	242: // Adding mover to group
		bWatchDogActive := TRUE;
		THIS^.fbMoversPresent.ResetIterator();
		WHILE THIS^.fbMoversPresent.HasNextObject() DO
			IF ToXpMover(THIS^.fbMoversPresent.GetNextObject(),ipTempMover) THEN
				hr := GetMostSignificant(hr, ipTempMover.Feedback.HR);
			END_IF
		END_WHILE
		
		IF CheckOk(hr) THEN 
			nSeqEnabling := 300;
		ELSIF FAILED(hr) THEN
			nSeqEnabling := 1000 + nSeqEnabling;
		END_IF		
	
		
		
	300: // Enable group
		bWatchDogActive := TRUE;
		hr := ipGroup.Enable();
		
		IF CheckOk(hr) THEN 
			nSeqEnabling := 310;
		ELSE
			nSeqEnabling := 1000 + nSeqEnabling;
		END_IF	
		
	310: // Enabling group
		bWatchDogActive := TRUE;
		hr := ipGroup.Feedback.HR;
		
		IF CheckOk(hr) THEN 
			//nSeqEnabling := 350;
			nSeqEnabling := 400;
		ELSIF FAILED(hr) THEN
			nSeqEnabling := 1000 + nSeqEnabling;
		END_IF	
		
		
//	340: // Check dist last known position to current pos
//		bWatchDogActive := TRUE;
//		THIS^.fbMovers.ResetIterator();
//		WHILE THIS^.fbMovers.HasNextObject() DO
//			IF ToXpMover(THIS^.fbMovers.GetNextObject(),ipTempMover) THEN
//				IF ipTempMover.PositionAtDisable.x <> 0 AND ipTempMover.PositionAtDisable.y <> 0 THEN
//					fDistLastToSet := F_DistXYVectors(ipTempMover.PositionAtDisable, ipTempMover.PositionSet);
//					fMaxError := MAX(fMaxError, fDistLastToSet);
//				END_IF
//			END_IF
//		END_WHILE
//		IF fMaxError < 50 THEN
//			nSeqEnabling := 350;
//		ELSE
//			nSeqEnabling := 400;			
//		END_IF
//
//		
//	350: // Move to last valide known position
//		bWatchDogActive := TRUE;
//		THIS^.fbMovers.ResetIterator();
//		WHILE THIS^.fbMovers.HasNextObject() DO
//			IF ToXpMover(THIS^.fbMovers.GetNextObject(),ipTempMover) THEN
//				IF ipTempMover.PositionAtDisable.x <> 0 AND ipTempMover.PositionAtDisable.y <> 0 THEN
//					hr := GetMostSignificant(hr, ipTempMover.MoveXY(fPosition_X := ipTempMover.PositionAtDisable.x, 
//																	fPosition_Y := ipTempMover.PositionAtDisable.y));
//				END_IF
//			END_IF
//		END_WHILE
//		//Its posible that the command failed. Do not exit SEQ
//		nSeqEnabling := 351;
//
//
//		
//	351: // Wait for standstill
//		bWatchDogActive := TRUE;
//		
//		bOk := TRUE;
//		THIS^.fbMovers.ResetIterator();
//		WHILE THIS^.fbMovers.HasNextObject() DO
//			IF ToXpMover(THIS^.fbMovers.GetNextObject(),ipTempMover) THEN
//				bOk := bOk AND ipTempMover.Standstill;
//			END_IF
//		END_WHILE
//		THIS^.fbMovers.RestoreIterator();
//		
//		IF bOk THEN 
//			nSeqEnabling := 400;
//		END_IF	

		
	400: (*	Restart of the sequenze "JoiningTrack". Default strategy is that each mover joins the closest track
			Outsourced to a method for easier overwriting *)
		THIS^.nSeqJoiningTrack := 0;	
		nSeqEnabling := 401;
	

	401: (*	Default strategy is that each mover joins the closest track
			Outsourced to a method for easier overwriting *)
		hr := THIS^.JoiningTrack();

		IF CheckOk(hr) THEN 
			nSeqEnabling := 500;
		ELSIF FAILED(hr) THEN
			nSeqEnabling := 1000 + nSeqEnabling;
		END_IF	
		
	

	
	500: (*	Restart of the sequenze "JoiningStation" to distribute the movers to the available stations.
			Outsourced to a method for easier overwriting *)
		THIS^.nSeqJoiningStation := 0;	
		nSeqEnabling := 501;	
	
	501: (*	Distribute the movers to the available stations.
		 	Outsourced to a method for easier overwriting *)
		hr := THIS^.JoiningStation();

		IF CheckOk(hr) THEN 
			nSeqEnabling := SEQ_DONE;
		ELSIF FAILED(hr) THEN
			nSeqEnabling := 1000 + nSeqEnabling;
		END_IF	

		
	SEQ_DONE: // Done
		Enabling := S_OK;

		
	1000..1999://Error
		hr := GetMostSignificant(hrLastCycle, E_FAIL);
		//Only rais if timeout is not active
		IF NOT fbErrorEnabling.bRaised AND NOT fbTimeOutEnabling.bRaised THEN 
			fbErrorEnabling.CreateEx(stEventEntry:=TC_EVENTS.CHALET_Base_Events.ErrorEnabling, ipSourceInfo := THIS^.fbSourceInfo, bWithConfirmation := FALSE);
			fbErrorEnabling.ipArguments.AddUInt(nSeqEnabling-1000);
			fbErrorEnabling.Raise(0);
		END_IF
	
	ELSE
		//Timeout unknown state
		bWatchDogActive := TRUE;
END_CASE


//Timeout after to long stay in one of the following seq.
fbTimeOutSeq.IN := (nlastState = nSeqEnabling) AND bWatchDogActive;
fbTimeOutSeq.PT := TO_TIME(XPlanarParameterlist.F_TIMEOUT_ERROR_ENABLING*1000.0);
fbTimeOutSeq();
nlastState := nSeqEnabling;

IF fbTimeOutSeq.Q THEN
	IF NOT fbTimeOutEnabling.bRaised THEN 
		fbTimeOutEnabling.CreateEx(stEventEntry:=TC_EVENTS.CHALET_Base_Events.TimeOutEnabling, ipSourceInfo := THIS^.fbSourceInfo, bWithConfirmation := FALSE);
		fbTimeOutEnabling.ipArguments.AddUInt(nSeqEnabling);
		fbTimeOutEnabling.Raise(0);
	END_IF
	//next seq is error
	nSeqEnabling := 1000 + nSeqEnabling;
END_IF

//Clear Tc3-Eventlogger alarm 
IF nSeqEnabling <= SEQ_DONE THEN
	fbTimeOutEnabling.Clear(0,0);
	fbErrorEnabling.Clear(0,0);
	fbErrorMoverDetection.Clear(0,0);
END_IF


//store last information
hrLastCycle := hr;

// Propagate error
IF FAILED(hr) THEN
	Enabling := hr;
END_IF
END_METHOD

{attribute 'monitoring':='call'}
PROPERTY Enviroment : I_XP_Environment
GET
Enviroment := THIS^.ipEnvironment;
END_GET
END_PROPERTY

METHOD FastStop : I_CH_Feedback
VAR
	ipMoverPlc : I_XP_Mover_PLC;
END_VAR
THIS^.MoversPresent.ResetIterator();
WHILE THIS^.MoversPresent.HasNextObject() DO
	IF __QUERYINTERFACE(THIS^.MoversPresent.GetNextObject(),ipMoverPlc) THEN
		//Change deceleration to MC_MAXIMUM for each mover
		ipMoverPlc.SetDynConstraint_Path(V:= MC_DEFAULT, A:= MC_DEFAULT, D:= MC_MAXIMUM, J:= MC_MAXIMUM);
	END_IF
END_WHILE
THIS^.MoversPresent.RestoreIterator();


FastStop := THIS^.Disable();
THIS^.Disabling();
END_METHOD

METHOD FB_init : BOOL
VAR_INPUT
	bInitRetains : BOOL; // if TRUE, the retain variables are initialized (warm start / cold start)
	bInCopyCode : BOOL;  // if TRUE, the instance afterwards gets moved into the copy code (online change)
	
END_VAR
VAR
	fbGetCurTaskIdx  : GETCURTASKINDEX;
END_VAR
THIS^.fbFeedback.ActiveCommand 		:= TO_STRING(THIS^.eActiveCommand);
END_METHOD

{attribute 'monitoring':='call'}
PROPERTY Feedback : CHALET_BaseComponents.I_CH_Feedback
GET
Feedback := THIS^.fbFeedback;
END_GET
END_PROPERTY

//Returns the station that is closest to the point according to Phytagoras
METHOD GetStationClosestTo : I_XP_Station
VAR_INPUT
	pos : MoverVector;
END_VAR
VAR
	stPositionStation : MoverVector;
	ipEachStation : I_XP_Station;
	fTempDist : LREAL;
	fDistClosestStation: LREAL := CHALET_BaseComponents.GVL_Datatypes.cMaxLreal;
END_VAR
THIS^.fbStationsUsed.ResetIterator();
WHILE THIS^.fbStationsUsed.HasNextObject() DO
	IF __QUERYINTERFACE(THIS^.fbStationsUsed.GetNextObject(),ipEachStation) THEN
		stPositionStation.x := ipEachStation.PositionOnTrackXY.x;
		stPositionStation.y := ipEachStation.PositionOnTrackXY.y;
		
		fTempDist := F_DistXYVectors(pos, stPositionStation);
		
		IF fTempDist <= fDistClosestStation THEN
			fDistClosestStation := fTempDist;
			GetStationClosestTo := ipEachStation;
		END_IF
		
	END_IF
END_WHILE
THIS^.fbStationsUsed.RestoreIterator();
END_METHOD

METHOD Initialize : HRESULT
VAR_INPUT
END_VAR
VAR
	hr 				: HRESULT := S_OK;
	ipEachStation 	: I_XP_Station;
END_VAR
VAR_INST
	//This error cannot be reset. Requires a reset cold
	{attribute 'hide'}	
	fbInitError : FB_TcAlarm;
	{attribute 'hide'}	
	fbMissingInterfaceAlarm : FB_TcAlarm;

END_VAR
//Set to busy on first call
IF THIS^.eActiveCommand <> CHALET_NC.E_NcAxisCommands.Initialize THEN
	THIS^.eActiveCommand 					:= CHALET_NC.E_NcAxisCommands.Initialize;
	THIS^.fbFeedback.ActiveCommand 			:= TO_STRING(THIS^.eActiveCommand);	
	THIS^.fbFeedback.LastCommandAccepted	:= TRUE;		
	THIS^.fbFeedback.Busy 					:= TRUE;
END_IF

//Check Error during FB_Init
IF THIS^.bErrorDuringFbInit THEN
	IF NOT fbInitError.bRaised THEN 
		//This error cannot be reset. Requires a reset cold
		fbInitError.CreateEx(stEventEntry:=TC_EVENTS.CHALET_Base_Events.ErrorFBinit, ipSourceInfo := THIS^.fbSourceInfo, bWithConfirmation := FALSE);
		fbInitError.Raise(0);
	END_IF
	Initialize:= E_FAIL;
	THIS^.fbFeedback.HR := Initialize;
	RETURN;
END_IF	


//Check if Envirement and Group is existing
IF  THIS^.ipGroup = 0 THEN
	IF NOT fbMissingInterfaceAlarm.bRaised THEN 
		//This error cannot be reset. Requires a reset cold
		fbMissingInterfaceAlarm.CreateEx(stEventEntry:=TC_EVENTS.CHALET_XPlanar_Events.MissingGroupe, ipSourceInfo := THIS^.fbSourceInfo, bWithConfirmation := FALSE);
		fbMissingInterfaceAlarm.Raise(0);
	END_IF
	Initialize := E_FAIL;
	THIS^.fbFeedback.HR := Initialize;
	RETURN;
END_IF

//Check if Envirement and Group is existing
IF THIS^.ipEnvironment = 0 THEN
	IF NOT fbMissingInterfaceAlarm.bRaised THEN 
		//This error cannot be reset. Requires a reset cold
		fbMissingInterfaceAlarm.CreateEx(stEventEntry:=TC_EVENTS.CHALET_XPlanar_Events.MissingEnvironment, ipSourceInfo := THIS^.fbSourceInfo, bWithConfirmation := FALSE);
		fbMissingInterfaceAlarm.Raise(0);
	END_IF
	Initialize := E_FAIL;
	THIS^.fbFeedback.HR := Initialize;
	RETURN;
END_IF



//Init envirement first to get access to XPlanar_Utility
IF THIS^.ipEnvironment.Initialize() = S_OK THEN
	hr := GetMostSignificant(hr, THIS^.ipGroup.Initialize());
	hr := GetMostSignificant(hr, THIS^.fbMoversPresent.Initialize());
	hr := GetMostSignificant(hr, THIS^.fbTracks.Initialize());
	hr := GetMostSignificant(hr, THIS^.fbStationsAll.Initialize());
	hr := GetMostSignificant(hr, THIS^.fbTriggers.Initialize());
	hr := GetMostSignificant(hr, THIS^.fbZones.Initialize());
ELSE
	hr := S_PENDING;
END_IF	



THIS^.bInitDone := (hr = S_OK);

Initialize:= hr;

THIS^.fbFeedback.HR := Initialize;
END_METHOD

{attribute 'monitoring':='call'}
PROPERTY Initialized : BOOL
GET
Initialized := bInitDone;
END_GET
END_PROPERTY

METHOD PROTECTED JoiningStation : HRESULT
VAR
	hr : HRESULT;
	ipEachMover : I_XP_Mover;
	ipEachMoverPlc : I_XP_Mover_PLC;
	ipEachMoverInStation : I_XP_Mover;
	ipEachStation : I_XP_Station;
	ipFirstStation : I_XP_Station;
	ipParentStation : I_XP_Station;
	ipTempMoverPlc : I_XP_Mover_PLC;

	//during move on track
	fVelo	: Tc3_Mc3Definitions.MC_LREAL := Tc3_Mc3Definitions.MC_DEFAULT; 
	fAccDec	: Tc3_Mc3Definitions.MC_LREAL := Tc3_Mc3Definitions.MC_DEFAULT;
	bError : BOOL;
	bFound : BOOL;
	bMoverAtCmdPos : BOOL;
	refPosition : REFERENCE TO MoverVector;
	fCalcualtedGapAtMoverPosition : LREAL;

	ipClosestStation : I_XP_Station;
	fDistToStation : LREAL := CHALET_BaseComponents.GVL_Datatypes.cMaxLreal;
END_VAR
VAR_INST
	bResetMovers : BOOL;	

	{attribute 'hide'}	
	fbDelayJoiningStation : TON;
END_VAR
CASE nSeqJoiningStation OF

	0: //Init
		fbDelayJoiningStation.IN := FALSE;
		
		IF fbStationsUsed.IsEmpty THEN
			nSeqJoiningStation := SEQ_DONE;
		ELSE
			nSeqJoiningStation := 10;
		END_IF
	


	
		
	10:	// For each Mover, Clear planed route to target. After enabling the tracks may have change and are not longer existing.
		THIS^.fbMoversPresent.ResetIterator();
		WHILE THIS^.fbMoversPresent.HasNextObject() DO
			IF __QUERYINTERFACE(THIS^.fbMoversPresent.GetNextObject(), ipEachMover) THEN
				//clear route
				ipEachMover.SetRouteToParent(0);
			END_IF
		END_WHILE
		THIS^.fbMoversPresent.RestoreIterator();
		
		//Empty Mover queue in station
		THIS^.fbStationsUsed.ResetIterator();
		WHILE THIS^.fbStationsUsed.HasNextObject() DO
			IF __QUERYINTERFACE(THIS^.fbStationsUsed.GetNextObject(), ipEachStation) THEN
				ipEachStation.DeleteMoversQueue(); // This is also reset the parent of each mover
			END_IF
		END_WHILE
		THIS^.fbStationsUsed.RestoreIterator();
		
		nSeqJoiningStation := 20;
	
	


	
		
	20: (*Check whether the last set station parent (station responsible for continuing to send the mover) is still valid. This is not the case if, for example:
		- Mover was manually moved to a new position
		- Track layout has changed
		- Position of the station has changed - No longer exists	*)
		THIS^.fbMoversPresent.ResetIterator();
		WHILE THIS^.fbMoversPresent.HasNextObject() DO
			IF __QUERYINTERFACE(THIS^.fbMoversPresent.GetNextObject(), ipEachMover) THEN
				//Prio 1: If the station ahead was the parent, kept this as parent. Easily accessible without issues with collision prevention
				ipParentStation := ipEachMover.CurrentTrack.StationAhedPosition(ipEachMover.PositionOnTrack);
				IF ipEachMover.LastValidParentStation = ipParentStation AND ipParentStation <> 0 THEN
					//Set as new parent
					ipParentStation.AddMoverToQueue(ipEachMover);
					CONTINUE; //Check next mover
				END_IF
				
				//Prio 2: If the station closest was the parent, +/- 10mm . Maybe mall issues with collision prevention
				ipParentStation := ipEachMover.CurrentTrack.StationClosestTo(ipEachMover.PositionOnTrack);
				fDistToStation := F_DistXYVectors(ipParentStation.PositionOnTrackXYZABC, ipEachMover.PositionSet);
				IF ipEachMover.LastValidParentStation = ipParentStation AND ipParentStation <> 0 AND fDistToStation < 10.0 THEN
					//Set as new parent
					ipParentStation.AddMoverToQueue(ipEachMover);
					CONTINUE; //Check next mover
				END_IF
				
				//Prio 3: Get any station ahead current position
				ipParentStation := ipEachMover.CurrentTrack.StationAhedPosition(ipEachMover.PositionOnTrack);
				//Set as new parent
				ipParentStation.AddMoverToQueue(ipEachMover);
			END_IF
		END_WHILE
		THIS^.fbMoversPresent.RestoreIterator();	
	
		nSeqJoiningStation := 30;	
	
	
	
	30: //Send Movers to parent - shortest way
		THIS^.fbMoversPresent.ResetIterator();
		WHILE THIS^.fbMoversPresent.HasNextObject() DO
			//Do for all Movers whitout a target station
			IF ToXpMover(THIS^.fbMoversPresent.GetNextObject(),ipEachMover) AND_THEN (ipEachMover.ParentStation <> 0) AND_THEN __QUERYINTERFACE(ipEachMover,ipEachMoverPlc) THEN
				//Set Path dynamic constraint to settings in XPlanarParameterlist. 0=Defalt
				IF XPlanarParameterlist.F_ENABLING_ON_TRACK_VELOCITY <> 0 THEN fVelo := XPlanarParameterlist.F_ENABLING_ON_TRACK_VELOCITY;END_IF
				IF XPlanarParameterlist.F_ENABLING_ON_TRACK_ACC_DEC <> 0 THEN fAccDec := XPlanarParameterlist.F_ENABLING_ON_TRACK_ACC_DEC;END_IF
			
				//Increase or decrease the mover DynConstraint for approaching the station 
				ipEachMoverPlc.SetDynConstraint_Path(	V:= fVelo, 
														A:= fAccDec, 
														D:= fAccDec, 
														J:= Tc3_Mc3Definitions.MC_DEFAULT);
		
				// gap depending on current position
				fCalcualtedGapAtMoverPosition := ipEachMover.CurrentTrack.GapAtPosition(ipEachMover.PositionOnTrack);
		
				hr := GetMostSignificant(hr, ipEachMover.MoveOnTrack_ShortestWay(ipTrack := ipEachMover.ParentStation.AccocietedTrack,
																				fPosition := ipEachMover.ParentStation.PositionOnTrack, 
																				fGap := fCalcualtedGapAtMoverPosition));
				
					
				END_IF
		END_WHILE
		THIS^.fbMoversPresent.RestoreIterator();		

		IF CheckOk(hr) THEN 
			nSeqJoiningStation := 100;
		ELSIF FAILED(hr) THEN
			nSeqJoiningStation := 1000 + nSeqJoiningStation;
		END_IF	
	
	
		
	100: //Delay to allow the movers to start movement
		fbDelayJoiningStation.IN := TRUE;
		fbDelayJoiningStation.PT := T#100MS;
		IF fbDelayJoiningStation.Q THEN
			nSeqJoiningStation := 110;
			fbDelayJoiningStation.IN := FALSE;
		END_IF
	
	
	110: //Wait for all movers until the movement is completed(speed =0)
		THIS^.fbMoversPresent.ResetIterator();
		WHILE THIS^.fbMoversPresent.HasNextObject() DO
			IF ToXpMover(THIS^.fbMoversPresent.GetNextObject(),ipEachMover) THEN
				//Check all movers if an error is active
				IF ipEachMover.Feedback.Error THEN
					hr := GetMostSignificant(hr, ipEachMover.Feedback.HR);
				//Wait for all movers to stop/finish movement
				ELSIF NOT (ipEachMover.Standstill) THEN
					hr := GetMostSignificant(hr, S_PENDING);
				END_IF
			END_IF
		END_WHILE 
		THIS^.fbMoversPresent.RestoreIterator();
		
		IF CheckOk(hr) THEN 
			nSeqJoiningStation := 500;
		ELSIF FAILED(hr) THEN
			nSeqJoiningStation := 1000 + nSeqJoiningStation;
		END_IF			

		
	500: // Check if a mover passes his parent station and is not abel to drive backwarts due to CA
		(* every mover who has not made it to his target position (presumably because of CA) gets a new parent station which is definitely in front and can therefore be reached.
			Blocked movers are thus released. This should have no effect on all other movers as the parent remains identical. *)
		
		//Empty Mover queue in station
		THIS^.fbStationsUsed.ResetIterator();
		WHILE THIS^.fbStationsUsed.HasNextObject() DO
			IF __QUERYINTERFACE(THIS^.fbStationsUsed.GetNextObject(), ipEachStation) THEN
				ipEachStation.DeleteMoversQueue(); // This is also reset the parent of each mover
			END_IF
		END_WHILE
		THIS^.fbStationsUsed.RestoreIterator();

		//Set first station ahead as target or set again last valide station
		THIS^.fbMoversPresent.ResetIterator();
		WHILE THIS^.fbMoversPresent.HasNextObject() DO
			IF ToXpMover(THIS^.fbMoversPresent.GetNextObject(),ipEachMover) THEN
				refPosition REF= ipEachMover.LastValidParentStation.PositionOnTrackXYZABC;
				bMoverAtCmdPos := F_DistXYVectors(ipEachMover.PositionSet, refPosition) < 1.0;
				//Set again last parent
				IF bMoverAtCmdPos THEN
					ipEachMover.LastValidParentStation.AddMoverToQueue(ipEachMover);
				ELSE
					ipParentStation := ipEachMover.CurrentTrack.StationAhedPosition(ipEachMover.PositionOnTrack);
					ipParentStation.AddMoverToQueue(ipEachMover);
				END_IF
			END_IF
		END_WHILE 
		THIS^.fbMoversPresent.RestoreIterator();
		nSeqJoiningStation := 501;
		
		
	501: //Start movement - shortest way
		THIS^.fbMoversPresent.ResetIterator();
		WHILE THIS^.fbMoversPresent.HasNextObject() DO
			//Do for all Movers whitout a target station
			IF ToXpMover(THIS^.fbMoversPresent.GetNextObject(),ipEachMover) AND_THEN (ipEachMover.ParentStation <> 0) AND_THEN __QUERYINTERFACE(ipEachMover,ipEachMoverPlc) THEN
				//Set Path dynamic constraint to settings in XPlanarParameterlist. 0=Defalt
				IF XPlanarParameterlist.F_ENABLING_ON_TRACK_VELOCITY <> 0 THEN fVelo := XPlanarParameterlist.F_ENABLING_ON_TRACK_VELOCITY;END_IF
				IF XPlanarParameterlist.F_ENABLING_ON_TRACK_ACC_DEC <> 0 THEN fAccDec := XPlanarParameterlist.F_ENABLING_ON_TRACK_ACC_DEC;END_IF
			
				//Increase or decrease the mover DynConstraint for approaching the station 
				ipEachMoverPlc.SetDynConstraint_Path(	V:= fVelo, 
														A:= fAccDec, 
														D:= fAccDec, 
														J:= Tc3_Mc3Definitions.MC_DEFAULT);
		
				// gap depending on current position
				fCalcualtedGapAtMoverPosition := ipEachMover.CurrentTrack.GapAtPosition(ipEachMover.PositionOnTrack);
		
				hr := GetMostSignificant(hr, ipEachMover.MoveOnTrack_ShortestWay(ipTrack := ipEachMover.ParentStation.AccocietedTrack,
																				fPosition := ipEachMover.ParentStation.PositionOnTrack, 
																				fGap := fCalcualtedGapAtMoverPosition));
				
					
				END_IF
		END_WHILE
		THIS^.fbMoversPresent.RestoreIterator();		

		IF CheckOk(hr) THEN 
			nSeqJoiningStation := SEQ_DONE;
		ELSIF FAILED(hr) THEN
			nSeqJoiningStation := 1000 + nSeqJoiningStation;
		END_IF	

	SEQ_DONE:
		;
	
	1000..1999://Error
		hr := GetMostSignificant(hr, E_FAIL);
END_CASE

//Update
fbDelayJoiningStation();


//Return value
IF FAILED(hr) THEN 
	//Error
    JoiningStation := GetMostSignificant(hr, E_FAIL);
ELSIF (nSeqJoiningStation = SEQ_DONE) THEN
	//Done
    JoiningStation := S_OK;
ELSE
	//Busy
    JoiningStation := S_PENDING;;
END_IF
END_METHOD

METHOD PROTECTED JoiningTrack : HRESULT
VAR	
	hr : HRESULT;
	ipClosestTrack, ipLastTrack : I_XP_Track;	
	ipEachMover : I_XP_Mover;
	ipEachTrack : I_XP_Track;
	fDistance : LREAL;
	fShortestDistance : LREAL;
	fDistToLastValidPos : LREAL;
	bUseClosestTrack : BOOL;
END_VAR
CASE nSeqJoiningTrack OF

	0: //Init
		IF fbTracks.IsEmpty THEN
			nSeqJoiningTrack := SEQ_DONE;
		ELSE
			nSeqJoiningTrack := 10;
		END_IF

		
	10: //Last or Closest Track	
		//compare to the last valid position whether the mover is still unchanged on the tile. 
		//If there is only a small movement <5mm, an attempt is made to move to the last position. 
		//Otherwise the closest track is moved to
		THIS^.fbMoversPresent.ResetIterator();
		WHILE THIS^.fbMoversPresent.HasNextObject() DO
			IF ToXpMover(THIS^.fbMoversPresent.GetNextObject(),ipEachMover) THEN
				//Calculate distance
				fDistToLastValidPos := F_DistXYVectors(ipEachMover.LastValidPositionXYZABC, ipEachMover.PositionSet);
	
				IF fDistToLastValidPos > 5.0 OR ipEachMover.LastValidTrack = 0 THEN
					bUseClosestTrack := TRUE;
					EXIT;
				END_IF
	
			END_IF
		END_WHILE
		THIS^.fbMoversPresent.RestoreIterator();	
		
		
		IF bUseClosestTrack THEN
			//Closest
			nSeqJoiningTrack := 50;
		ELSE
			//Last
			nSeqJoiningTrack := 60;
		END_IF
		
		
		
	50:// Join closest track
		THIS^.fbMoversPresent.ResetIterator();
		WHILE THIS^.fbMoversPresent.HasNextObject() DO
			IF ToXpMover(THIS^.fbMoversPresent.GetNextObject(),ipEachMover) THEN
				
				//check all track to decide which is the closest
				//start with the greatest possible distance, so that each track is definitely closer
				fShortestDistance := CHALET_BaseComponents.GVL_Datatypes.cMaxLreal; 
				THIS^.fbTracks.ResetIterator();			
				WHILE THIS^.fbTracks.HasNextObject() DO
					IF ToXpTrack(THIS^.fbTracks.GetNextObject(),ipEachTrack) THEN
						fDistance := ipEachMover.DistToTrack(ipEachTrack);
						//closer track found
						IF fDistance <= fShortestDistance THEN
							ipClosestTrack := ipEachTrack;
							fShortestDistance := fDistance;
						END_IF
					END_IF
				END_WHILE
				THIS^.fbTracks.RestoreIterator();		
				

				IF ipClosestTrack <> 0 THEN
					hr := GetMostSignificant(hr, ipEachMover.JoinTrack(ipClosestTrack));
				ELSE
					hr := GetMostSignificant(hr, E_FAIL);
				END_IF
			
				
			END_IF
		END_WHILE
		THIS^.fbMoversPresent.RestoreIterator();
		nSeqJoiningTrack := 100;		
		
		
	60:// Move to last known position
		THIS^.fbMoversPresent.ResetIterator();
		WHILE THIS^.fbMoversPresent.HasNextObject() DO
			IF ToXpMover(THIS^.fbMoversPresent.GetNextObject(),ipEachMover) THEN
				hr := GetMostSignificant(hr, ipEachMover.MoveXY(ipEachMover.LastValidPositionXYZABC.x, ipEachMover.LastValidPositionXYZABC.y));
			END_IF
		END_WHILE
		THIS^.fbMoversPresent.RestoreIterator();
		nSeqJoiningTrack := 61;		
		
	61: // Moving check feedback
		THIS^.fbMoversPresent.ResetIterator();
		WHILE THIS^.fbMoversPresent.HasNextObject() DO
			IF ToXpMover(THIS^.fbMoversPresent.GetNextObject(),ipEachMover) THEN
				// Check mover errors
				hr := GetMostSignificant(hr, ipEachMover.Feedback.HR);
			END_IF
		END_WHILE
		THIS^.fbMoversPresent.RestoreIterator();		
		
		IF CheckOk(hr) THEN 
			nSeqJoiningTrack := 62;
		ELSIF FAILED(hr) THEN
			nSeqJoiningTrack := 1000 + nSeqJoiningTrack;
		END_IF	
		
	62: //Join last valid track
		THIS^.fbMoversPresent.ResetIterator();
		WHILE THIS^.fbMoversPresent.HasNextObject() DO
			IF ToXpMover(THIS^.fbMoversPresent.GetNextObject(),ipEachMover) THEN
				ipLastTrack := ipEachMover.LastValidTrack;
				hr := GetMostSignificant(hr, ipEachMover.JoinTrack(ipLastTrack));
			END_IF
		END_WHILE
		THIS^.fbMoversPresent.RestoreIterator();
		nSeqJoiningTrack := 100;
		
		
	100: // Joining  track check feedback
		THIS^.fbMoversPresent.ResetIterator();
		WHILE THIS^.fbMoversPresent.HasNextObject() DO
			IF ToXpMover(THIS^.fbMoversPresent.GetNextObject(),ipEachMover) THEN
				
				// Check mover errors
				hr := GetMostSignificant(hr, ipEachMover.Feedback.HR);
				
				//Check if Mover is on track
				IF NOT (ipEachMover.Mode = MC_PLANAR_MOVER_COMMAND_MODE.OnTrack) THEN
					hr := GetMostSignificant(hr, S_PENDING);
				END_IF
			END_IF
		END_WHILE
		THIS^.fbMoversPresent.RestoreIterator();
		
		IF CheckOk(hr) THEN 
			nSeqJoiningTrack := SEQ_DONE;
		ELSIF FAILED(hr) THEN
			nSeqJoiningTrack := 1000 + nSeqJoiningTrack;
		END_IF			

		
	1000..1999://Error
		hr := GetMostSignificant(hr, E_FAIL);
END_CASE

		
		
//Return value
IF FAILED(hr) THEN 
	//Error
    JoiningTrack := GetMostSignificant(hr, E_FAIL);
ELSIF (nSeqJoiningTrack = SEQ_DONE) THEN
	//Done
    JoiningTrack := S_OK;
ELSE
	//Busy
    JoiningTrack := S_PENDING;;
END_IF
END_METHOD

METHOD LinkEnvironment : HRESULT
VAR_INPUT
	ipEnvironment : I_CH_Object;
END_VAR

VAR
	ipXpEnvironment : I_XP_Environment;
END_VAR
IF ipEnvironment <> 0 AND_THEN __QUERYINTERFACE(ipEnvironment,ipXpEnvironment) THEN
	THIS^.ipEnvironment := ipXpEnvironment;
ELSE
	LinkEnvironment := E_FAIL;
	THIS^.bErrorDuringFbInit := TRUE;
END_IF
END_METHOD

METHOD LinkGroup : HRESULT
VAR_INPUT
	ipGroup : I_CH_Object;
END_VAR

VAR
	ipXpGroup : I_XP_Group;
END_VAR
IF ipGroup <> 0 AND_THEN __QUERYINTERFACE(ipGroup,ipXpGroup) THEN
	THIS^.ipGroup := ipXpGroup;
ELSE
	LinkGroup := E_FAIL;
	THIS^.bErrorDuringFbInit := TRUE;
END_IF
END_METHOD

{attribute 'monitoring':='call'}
//List of movers that are not present in the current system
PROPERTY MoversNotPresent : CHALET_BaseComponents.I_CH_LIST
GET
MoversNotPresent := THIS^.fbMoversNotPresent;
END_GET
END_PROPERTY

{attribute 'monitoring':='call'}
//List of movers that are present in the current system
PROPERTY MoversPresent : CHALET_BaseComponents.I_CH_LIST
GET
MoversPresent := THIS^.fbMoversPresent;
END_GET
END_PROPERTY

{attribute 'monitoring':='call'}
PROPERTY Paths : CHALET_BaseComponents.I_CH_LIST
GET
Paths := THIS^.fbPaths;
END_GET
END_PROPERTY

METHOD RegisterMover : HRESULT
VAR_INPUT
	ipMover : I_CH_Object;
END_VAR

VAR
	ipXpMover : I_XP_Mover;
END_VAR
IF ipMover = 0 THEN
	//Invalide interface	
	THIS^.bErrorDuringFbInit := TRUE;
	RegisterMover := E_FAIL;
	
ELSIF NOT __QUERYINTERFACE(ipMover, ipXpMover) THEN
	//The required interface is missing
	THIS^.bErrorDuringFbInit := TRUE;
	RegisterMover := E_FAIL;
	
ELSIF THIS^.fbMoversPresent.IsFull THEN
	//List is full
	THIS^.bErrorDuringFbInit := TRUE;
	RegisterMover := E_FAIL;
	
ELSIF THIS^.bInitDone THEN
	//To late. System is initilized
	THIS^.bErrorDuringFbInit := TRUE;
	RegisterMover := E_FAIL;
	
ELSE
	
	THIS^.fbMoversPresent.AddObject(ipMover);
END_IF
END_METHOD

METHOD RegisterStation : HRESULT
VAR_INPUT
	ipStation : I_CH_Object;
END_VAR

VAR
	ipXpStation : I_XP_Station;
END_VAR
IF ipStation = 0 THEN
	//Invalide interface	
	THIS^.bErrorDuringFbInit := TRUE;
	RegisterStation := E_FAIL;
	
ELSIF NOT __QUERYINTERFACE(ipStation, ipXpStation) THEN
	//The required interface is missing
	THIS^.bErrorDuringFbInit := TRUE;
	RegisterStation := E_FAIL;
	
ELSIF THIS^.fbStationsUsed.IsFull THEN
	//List is full
	THIS^.bErrorDuringFbInit := TRUE;
	RegisterStation := E_FAIL;
	
ELSIF THIS^.bInitDone THEN
	//To late. System is initilized
	THIS^.bErrorDuringFbInit := TRUE;
	RegisterStation := E_FAIL;
		
ELSE
	
	THIS^.fbStationsAll.AddObject(ipStation);
END_IF
END_METHOD

METHOD RegisterTrack : HRESULT
VAR_INPUT
	ipTrack : I_CH_Object;
END_VAR

VAR
	ipXpTrack : I_XP_Track;
END_VAR
IF ipTrack = 0 THEN
	//Invalide interface	
	THIS^.bErrorDuringFbInit := TRUE;
	RegisterTrack := E_FAIL;
	
ELSIF NOT __QUERYINTERFACE(ipTrack, ipXpTrack) THEN
	//The required interface is missing
	THIS^.bErrorDuringFbInit := TRUE;
	RegisterTrack := E_FAIL;
	
ELSIF THIS^.fbTracks.IsFull THEN
	//List is full
	THIS^.bErrorDuringFbInit := TRUE;
	RegisterTrack := E_FAIL;
	
ELSIF THIS^.bInitDone THEN
	//To late. System is initilized
	THIS^.bErrorDuringFbInit := TRUE;
	RegisterTrack := E_FAIL;
		
ELSE
	
	THIS^.fbTracks.AddObject(ipTrack);
END_IF
END_METHOD

METHOD RegisterTrigger : HRESULT
VAR_INPUT
	ipTrigger	: CHALET_BaseComponents.I_CH_Object;
END_VAR
VAR
	ipXpTrigger : I_Xp_Trigger;
END_VAR
IF ipTrigger = 0 THEN
	//Invalide interface	
	THIS^.bErrorDuringFbInit := TRUE;
	RegisterTrigger := E_FAIL;
	
ELSIF NOT __QUERYINTERFACE(ipTrigger, ipXpTrigger) THEN
	//The required interface is missing
	THIS^.bErrorDuringFbInit := TRUE;
	RegisterTrigger := E_FAIL;
	
ELSIF THIS^.fbTriggers.IsFull THEN
	//List is full
	THIS^.bErrorDuringFbInit := TRUE;
	RegisterTrigger := E_FAIL;
	
ELSIF THIS^.bInitDone THEN
	//To late. System is initilized
	THIS^.bErrorDuringFbInit := TRUE;
	RegisterTrigger := E_FAIL;
		
ELSE
	
	THIS^.fbTriggers.AddObject(ipTrigger);
END_IF
END_METHOD

METHOD RegisterZone : HRESULT
VAR_INPUT
	ipZone	: CHALET_BaseComponents.I_CH_Object;
END_VAR
VAR
	ipXpsZone : I_XP_Zone;
END_VAR
IF ipZone = 0 THEN
	//Invalide interface	
	THIS^.bErrorDuringFbInit := TRUE;
	RegisterZone := E_FAIL;

ELSIF NOT __QUERYINTERFACE(ipZone, ipXpsZone) THEN
	//The required interface is missing
	THIS^.bErrorDuringFbInit := TRUE;
	RegisterZone := E_FAIL;
	
ELSIF THIS^.fbZones.IsFull THEN
	//List is full
	THIS^.bErrorDuringFbInit := TRUE;
	RegisterZone := E_FAIL;
	
ELSIF THIS^.bInitDone THEN
	//To late. System is initilized
	THIS^.bErrorDuringFbInit := TRUE;
	RegisterZone := E_FAIL;
		
ELSE
	
	THIS^.fbZones.AddObject(ipZone);	
END_IF
END_METHOD

METHOD RemoveMoverFromSystem : HRESULT
VAR_INPUT
	ipMover : I_XP_Mover;
END_VAR

IF ipMover <> 0 THEN
	THIS^.fbMoversPresent.RemoveObject(ipMover);
	
	ipMover.Disassemble();
	
	
	//Add if not already in list
	IF NOT THIS^.fbMoversNotPresent.ObjectInList(ipMover) THEN
		THIS^.fbMoversNotPresent.AddObject(ipMover);
	END_IF
END_IF
END_METHOD

METHOD Station : I_XP_Station_PLC
VAR_INPUT
	sLUID : STRING;
END_VAR
//IF no station was found, INTERFACE is 0 -> can generate fatal error
__QUERYINTERFACE(THIS^.fbStationsUsed.FindLUID(sLUID),Station);
END_METHOD

{attribute 'monitoring':='call'}
//List of all station objects that exist in this project
PROPERTY StationsAll : CHALET_BaseComponents.I_CH_LIST
GET
StationsAll := THIS^.fbStationsAll;
END_GET
END_PROPERTY

{attribute 'monitoring':='call'}
//List of all station objects that are considered for path planning in the currently running system
PROPERTY StationsUsed : CHALET_BaseComponents.I_CH_LIST
GET
StationsUsed := THIS^.fbStationsUsed;
END_GET
END_PROPERTY

//Suppress to change the dynamic(Gap) of passing movers in all stations. This is usefull in startup
PROPERTY SuppressAllDynamicsChanges : BOOL
SET
VAR
	ipTempStationPlc : I_XP_Station_PLC;
END_VAR
// go through the list and write request to it
THIS^.fbStationsUsed.ResetIterator();
WHILE THIS^.fbStationsUsed.HasNextObject() DO
	IF __QUERYINTERFACE(THIS^.fbStationsUsed.GetNextObject(), ipTempStationPlc) THEN
		ipTempStationPlc.SuppressDynamicsChange := SuppressAllDynamicsChanges;
	END_IF
END_WHILE
THIS^.fbStationsUsed.RestoreIterator();
END_SET
END_PROPERTY

{attribute 'monitoring':='call'}
PROPERTY Tracks : CHALET_BaseComponents.I_CH_LIST
GET
Tracks := THIS^.fbTracks;
END_GET
END_PROPERTY

{attribute 'monitoring':='call'}
PROPERTY Triggers : CHALET_BaseComponents.I_CH_LIST
GET
Triggers := THIS^.fbTriggers;
END_GET
END_PROPERTY

METHOD Update : HRESULT
VAR
	hr : HRESULT;
END_VAR
//Force to do an init at beginn
IF NOT THIS^.Initialized THEN
	THIS^.Initialize();
	RETURN;
END_IF

hr := S_OK;

hr := GetMostSignificant(hr, THIS^.Enabling());
hr := GetMostSignificant(hr, THIS^.Disabling());




// ********************** Set feedback depending on active command *******************************
CASE THIS^.eActiveCommand OF
	E_NcAxisCommands.None: 
		;

	E_NcAxisCommands.Initialize:
		fbFeedback.Busy 		:= NOT THIS^.bInitDone;
		fbFeedback.Done 		:= THIS^.bInitDone;
		fbFeedback.ErrorId 		:= 0;
		
	E_NcAxisCommands.Enable:
		fbFeedback.Busy 		:= nSeqEnabling > 0;
		fbFeedback.Done 		:= THIS^.Enabled;
		IF nSeqEnabling > 1000 THEN
			fbFeedback.ErrorId 		:= nSeqEnabling;
		END_IF
		
	E_NcAxisCommands.Disable:
		fbFeedback.Busy 		:= nSeqDisabling > 0;
		fbFeedback.Done 		:= THIS^.Disabled;
		IF nSeqDisabling > 1000 THEN
			fbFeedback.ErrorId 		:= nSeqDisabling;
		END_IF
		


	ELSE//External command in subclass
		;
END_CASE


// **********************  Stop to execute commands on .done or .error ***************************
IF fbFeedback.Done OR THIS^.fbFeedback.Error THEN
	eActiveCommand 				:= E_NcAxisCommands.None;
END_IF

CheckForErrors();

hr := GetMostSignificant(hr, THIS^.fbMoversPresent.Update());
hr := GetMostSignificant(hr, THIS^.fbTracks.Update());
hr := GetMostSignificant(hr, THIS^.fbStationsUsed.Update());
hr := GetMostSignificant(hr, THIS^.fbZones.Update());
hr := GetMostSignificant(hr, THIS^.fbTriggers.Update());
hr := GetMostSignificant(hr, THIS^.ipGroup.Update());
hr := GetMostSignificant(hr, THIS^.ipEnvironment.Update());


Update:= hr;
END_METHOD

{attribute 'monitoring':='call'}
PROPERTY Zones : CHALET_BaseComponents.I_CH_LIST
GET
Zones := THIS^.fbZones;
END_GET
END_PROPERTY

END_FUNCTION_BLOCK

// ---- COMPONENTs/Track/FB_XP_Track.TcPOU
{attribute 'no_explicit_call' := 'Do not call the body - Stick to OOP'}
(* XPlanar track - n per associated XPlanar. Can be instantiated as an array and/or individually
	The Planar track is a software object that represents a (virtual) one-dimensional path on the two-dimensional XPlanar stator surface. 
	Several Planar movers can be lined up and moved on this path. Collisions are prevented by keeping a preset distance between the movers. *)	
FUNCTION_BLOCK FB_XP_Track EXTENDS FB_CH_Object IMPLEMENTS I_XP_Track
VAR
	//Link to Planar-Track object
	fbTrack : MC_PlanarTrack;
	
	{attribute 'hide'}  
	bInitDone : BOOL := FALSE;
	{attribute 'hide'}               	
	fbFeedback 			: FB_XP_Feedback(ipSourceInfo := fbSourceInfo);	
	{attribute 'hide'}                   	
	eActiveCommand 		: CHALET_Nc.E_NcAxisCommands := CHALET_Nc.E_NcAxisCommands.None;
	{attribute 'hide'}
	ipXpSystem : I_XP_System_Registration;
	{attribute 'hide'}	
	nSeqConfiguring : UINT;
	{attribute 'hide'} 
	ipTracksEndAtThis : ARRAY[0..(XPlanarParameterlist.N_MAX_STATIONS_AHEAD_OR_BEHIND-1)] OF I_XP_Track;
	{attribute 'hide'} 
	ipTracksStartFromThis : ARRAY[0..(XPlanarParameterlist.N_MAX_STATIONS_AHEAD_OR_BEHIND-1)] OF I_XP_Track;
	{attribute 'hide'}  
	fbListOfStationsOnTrack : FB_CH_List;

	{attribute 'hide'}  
	bIsClosedLoop : BOOL;
	{attribute 'hide'}  
	PreviousTrackOTCIDs 	: ARRAY[0..(XPlanarParameterlist.N_MAX_STATIONS_AHEAD_OR_BEHIND-1)] OF OTCID;
	{attribute 'hide'}  
	SubsequentTrackOTCIDs 	: ARRAY[0..(XPlanarParameterlist.N_MAX_STATIONS_AHEAD_OR_BEHIND-1)] OF OTCID;
	
	{attribute 'hide'}
	fbListOfMoversOnTrack : FB_CH_List;
	{attribute 'hide'}  
	fbTracksAhead : FB_CH_List;
	{attribute 'hide'}  
	fbTracksBehinde : FB_CH_List;
	

	{attribute 'hide'}  
	fbListPathsOnThisTrack : FB_CH_List;	
	//Interface to this track in XPlanar Utility Lib
	ipUtilityTrack  : Tc3_XPlanarUtility.I_McPlanarTrack;
	
	fbHelpferStationOnEndOfThisTrack : FB_XP_Station(	ipSystem 			:= 0,
														ipAccocietedTrack 	:= (THIS^),// =closest track
														sUniqueName			:= '',
														sTargetGroup		:= '',
														nMoverQueueSize		:= 0,
														xPos				:= 0,
														yPos				:= 0);	
														
	//MC_CIRCLE_XYC_START_CENTER_END has the size of 72 byte													
	aRawGeometricElements : ARRAY[0.. XPlanarParameterlist.N_MAX_GEOMETRIC_ELEMENTS_PER_TRACK *72] OF LREAL;
	//Interface to TcComTrack ObjectId
	ipComObject : ITComObject;
END_VAR
VAR CONSTANT
	N_IDX_OFFSET_PREVIOUS_TRACK 	: UDINT := 16#050300D5; // Parameter(online) in Planar Track object
	N_IDX_OFFSET_SUBSEQUENT_TRACK 	: UDINT := 16#050300D6; // Parameter(online) in Planar Track object	
	N_IDX_OFFSET_IS_CLOSED_LOOP		: UDINT := 16#050300E1; // Parameter(online) in Planar Track object	
	N_IDX_GEOMETRIC_INFO			: UDINT := 16#050300D7; // Parameter(offline) in Planar Track object	
	GUID_MC_CIRCLE_XYC_START_CENTER_END			: GUID := Tc2_Utilities.STRING_TO_GUID(in:= 'C3BAEC31-7F05-4B2F-A9AE-F0D8872EE557');
	GUID_MC_POINT_XYC 							: GUID := Tc2_Utilities.STRING_TO_GUID(in:= '9E820E67-264A-4170-958A-0B26CA5C91FA');
	GUID_MC_LINE_XYC 							: GUID := Tc2_Utilities.STRING_TO_GUID(in:= 'B48A64D8-464F-4B39-8708-C82C1147C8B6');
END_VAR


// Planar-Feedback objects
VAR
	{attribute 'hide'} 
	fbFeedbackDisable		: MC_PlanarFeedback;
	{attribute 'hide'} 
	fbFeedbackEnable 		: MC_PlanarFeedback;
	{attribute 'hide'} 
	fbFeedbackAddToGrp 		: MC_PlanarFeedback;
	{attribute 'hide'} 
	fbFeedbackRmvFromGrp 	: MC_PlanarFeedback;
	{attribute 'hide'} 
	fbFeedbackReset 		: MC_PlanarFeedback;
END_VAR

METHOD AddMover : HRESULT
VAR_INPUT
	ipMover : I_XP_Mover;
END_VAR
IF ipMover <> 0 THEN
	AddMover := ipMover.JoinTrack(THIS^);
ELSE
	AddMover := E_FAIL;
END_IF
END_METHOD

METHOD AddToGroup : HRESULT
VAR_INPUT
	iGroup : I_XP_Group;
END_VAR
IF NOT THIS^.fbFeedback.Busy THEN
	THIS^.eActiveCommand 				:= CHALET_NC.E_NcAxisCommands.AddToGroupe;
	THIS^.fbFeedback.ActiveCommand 		:= TO_STRING(THIS^.eActiveCommand);	
	THIS^.fbFeedback.LastCommandAccepted:= TRUE;		
	THIS^.fbFeedback.Busy 				:= TRUE;
	
	iGroup.AddTrack(THIS^.fbTrack, THIS^.fbFeedbackAddToGrp);
	AddToGroup := S_OK;
ELSE
	AddToGroup := S_FALSE;
	THIS^.fbFeedback.LastCommandAccepted:= FALSE;	
END_IF
END_METHOD

{attribute 'monitoring':='call'}
PROPERTY ClosedLoop : BOOL
GET
ClosedLoop := bIsClosedLoop;
END_GET
END_PROPERTY

METHOD Configure : HRESULT // This is called once during system enabling
VAR_INPUT
END_VAR
VAR_INST
	{attribute 'hide'}  
	fbAlarmTrackLength0 : FB_TcAlarm;
END_VAR
// Validate settings
IF THIS^.Length = 0 THEN
	Configure := E_FAIL;
	THIS^.fbFeedback.LastCommandAccepted:= FALSE;	
	IF NOT fbAlarmTrackLength0.bRaised THEN
		fbAlarmTrackLength0.CreateEx(stEventEntry:= TC_EVENTS.CHALET_XPlanar_Events.TrackLength0, bWithConfirmation := FALSE, ipSourceInfo := THIS^.fbSourceInfo);
		fbAlarmTrackLength0.Raise(0);
	END_IF
	RETURN;
ELSE
	fbAlarmTrackLength0.Clear(0,0);	
END_IF



THIS^.eActiveCommand 				:= CHALET_NC.E_NcAxisCommands.Configure;
THIS^.fbFeedback.ActiveCommand 		:= TO_STRING(THIS^.eActiveCommand);	
THIS^.fbFeedback.LastCommandAccepted:= TRUE;		
THIS^.fbFeedback.Busy 				:= TRUE;

THIS^.nSeqConfiguring := 10;
Configure := S_OK;
END_METHOD

METHOD Configuring : HRESULT // This is called until S_OK during system enabling
VAR
	ipEachTrackObj : I_CH_Object;
	nIdx : UDINT;
	ipTrackComObject : ITComObject;
	nParaSize : UDINT;
	pParaData : PVOID;
	hr : HRESULT;
END_VAR
Configuring := S_PENDING;
CASE nSeqConfiguring OF
	0: // Idle
		Configuring := S_OK;
		
	10: //Start
		nSeqConfiguring := 200;
		
		
		
	200: //Read information from Track TcCom object
		//Get interface to ComObject
		FW_ObjMgr_GetObjectInstance(oid:= THIS^.OID, iid:= TC_GLOBAL_IID_LIST.IID_ITComObject, pipUnk:= ADR(ipTrackComObject));
	
		IF ipTrackComObject = 0 THEN
			//Error, interface not found
			nSeqConfiguring := nSeqConfiguring + 1000;	
		ELSE
			//Read array of oids PreviousTrackOTCIDs
			nParaSize := SIZEOF(THIS^.PreviousTrackOTCIDs);	pParaData := ADR(THIS^.PreviousTrackOTCIDs);
			hr := ipTrackComObject.TcGetObjPara(pid:=N_IDX_OFFSET_PREVIOUS_TRACK , nData:= nParaSize, pData:= pParaData, pgp:=0 );
			
			//Read array of oids SubsequentTrackOTCIDs
			nParaSize := SIZEOF(THIS^.SubsequentTrackOTCIDs);	pParaData := ADR(THIS^.SubsequentTrackOTCIDs);
			hr := ipTrackComObject.TcGetObjPara(pid:=N_IDX_OFFSET_SUBSEQUENT_TRACK , nData:= nParaSize, pData:= pParaData, pgp:=0 );			
			
			//Read bool CLOSED_LOOP
			nParaSize := SIZEOF(THIS^.bIsClosedLoop);	pParaData := ADR(THIS^.bIsClosedLoop);
			hr := ipTrackComObject.TcGetObjPara(pid:=N_IDX_OFFSET_IS_CLOSED_LOOP , nData:= nParaSize, pData:= pParaData, pgp:=0 );		
			FW_SafeRelease(ADR(ipTrackComObject));

			nSeqConfiguring := 300;
		END_IF
		
			
	300: // Convert SubsequentTrackOTCIDs to I_XP_Track and add to fbTracksAhead
		fbTracksAhead.Clear();
		FOR nIdx := 0 TO (XPlanarParameterlist.N_MAX_STATIONS_AHEAD_OR_BEHIND-1) DO
			//Get interface to object
			ipEachTrackObj := THIS^.ipXpSystem.Tracks.FindOID(THIS^.SubsequentTrackOTCIDs[nIdx]);
			//convert object -> I_XP_Track. If found, store in list
			IF ToXpTrack(ipEachTrackObj, ipTracksStartFromThis[nIdx]) THEN
				fbTracksAhead.AddObject(ipEachTrackObj);
				
			ELSIF THIS^.SubsequentTrackOTCIDs[nIdx] = 0 THEN
				;//No OTCID
				
			ELSE
				//Error, no track found with following oid
				nSeqConfiguring := nSeqConfiguring + 1000;	
				RETURN;;				
			END_IF
		END_FOR
		nSeqConfiguring := 301;		
	

	301: // Convert PreviousTrackOTCIDs to I_XP_Track and add to fbTracksBehinde
		fbTracksBehinde.Clear();
		FOR nIdx := 0 TO (XPlanarParameterlist.N_MAX_STATIONS_AHEAD_OR_BEHIND-1) DO
			//Get interface to object
			ipEachTrackObj := THIS^.ipXpSystem.Tracks.FindOID(THIS^.PreviousTrackOTCIDs[nIdx]);
			//convert object -> I_XP_Track. If found, store in list
			IF ToXpTrack(ipEachTrackObj, ipTracksEndAtThis[nIdx]) THEN
				fbTracksBehinde.AddObject(ipEachTrackObj);
				
			ELSIF THIS^.PreviousTrackOTCIDs[nIdx] = 0 THEN
				;//No OTCID
				
			ELSE
				//Error, no track found with following oid
				nSeqConfiguring := nSeqConfiguring + 1000;	
				RETURN;;				
			END_IF
		END_FOR			
		nSeqConfiguring := 400;

		
	400: //Configure the helper station who is located at the end of this track to improve komplex track routing
		THIS^.fbHelpferStationOnEndOfThisTrack.PositionXY.SetValuesXY(THIS^.EndPosition.x, THIS^.EndPosition.y);
		THIS^.fbHelpferStationOnEndOfThisTrack.SuppressDynamicsChange := TRUE;
		nSeqConfiguring := 999;

		
	
	999: // Done
		Configuring := S_OK;
		
	1000..1999://Error
		Configuring := E_FAIL;
END_CASE
END_METHOD

{attribute 'monitoring':='call'}
PROPERTY CtsMoversOnTrack : UINT
GET
THIS^.Prepare();//Prepare a list movers on this track


CtsMoversOnTrack := TO_UINT(THIS^.fbListOfMoversOnTrack.Size);
END_GET
END_PROPERTY

METHOD Disable : HRESULT
VAR_INPUT
END_VAR
IF NOT THIS^.fbFeedback.Busy THEN
	THIS^.eActiveCommand 				:= CHALET_NC.E_NcAxisCommands.Disable;
	THIS^.fbFeedback.ActiveCommand 		:= TO_STRING(THIS^.eActiveCommand);	
	THIS^.fbFeedback.LastCommandAccepted:= TRUE;		
	THIS^.fbFeedback.Busy 				:= TRUE;

	THIS^.fbTrack.Disable(fbFeedbackDisable);
	Disable := S_OK;
ELSE
	Disable := S_FALSE;
	THIS^.fbFeedback.LastCommandAccepted:= FALSE;	
END_IF
END_METHOD

METHOD Enable : HRESULT
VAR_INPUT
END_VAR
IF NOT THIS^.fbFeedback.Busy THEN
	THIS^.eActiveCommand 				:= CHALET_NC.E_NcAxisCommands.Enable;
	THIS^.fbFeedback.ActiveCommand 		:= TO_STRING(THIS^.eActiveCommand);	
	THIS^.fbFeedback.LastCommandAccepted:= TRUE;		
	THIS^.fbFeedback.Busy 				:= TRUE;

	THIS^.fbTrack.Enable(fbFeedbackEnable);
	Enable := S_OK;
ELSE
	Enable := S_FALSE;
	THIS^.fbFeedback.LastCommandAccepted:= FALSE;	
END_IF
END_METHOD

{attribute 'monitoring':='call'}
//Position of the end point of this tracks
PROPERTY EndPosition : REFERENCE TO MoverVector
GET
VAR_INST
	stEndPositionXY : MoverVector;
END_VAR
VAR
	fbPositionXYC : PositionXYC;
END_VAR
THIS^.fbTrack.GetPositionAt(THIS^.Length,fbPositionXYC);


stEndPositionXY.x := fbPositionXYC.x;
stEndPositionXY.y := fbPositionXYC.y;
stEndPositionXY.z := 0;
stEndPositionXY.a := 0;
stEndPositionXY.b := 0;
stEndPositionXY.c := fbPositionXYC.c;



EndPosition REF= stEndPositionXY;
END_GET
END_PROPERTY

METHOD FB_exit : BOOL
VAR_INPUT
	bInCopyCode : BOOL; // if TRUE, the exit method is called for exiting an instance that is copied afterwards (online change).
END_VAR

FW_SafeRelease(ADR(THIS^.ipComObject));
END_METHOD

METHOD FB_init : BOOL
VAR_INPUT
	bInitRetains : BOOL; // if TRUE, the retain variables are initialized (warm start / cold start)
	bInCopyCode : BOOL;  // if TRUE, the instance afterwards gets moved into the copy code (online change)
	
	ipSystem : I_CH_Object;
END_VAR
//Do the following code once during start up and not during onlinechange
IF NOT bInCopyCode THEN 
	
	(* Register to the Xplanar System
	   1. Test if the interface exists
	   2. Test if the object implements a "System for Mover" interface 
	*)
	IF ipSystem <> 0 AND_THEN __QUERYINTERFACE(ipSystem,THIS^.ipXpSystem) THEN
		THIS^.ipXpSystem.RegisterTrack(THIS^);
		
		
		THIS^.fbHelpferStationOnEndOfThisTrack.FB_init(	bInCopyCode			:= FALSE,
														bInitRetains		:= bInitRetains,
														ipSystem 			:= ipSystem,
														ipAccocietedTrack 	:= (THIS^),// =closest track
														sUniqueName			:= CONCAT('HelperStationAtEndOf', THIS^.LUID),
														sTargetGroup		:= '',
														nMoverQueueSize		:= 0,
														xPos				:= 0,
														yPos				:= 0);	
	END_IF

	THIS^.fbFeedback.ActiveCommand 		:= TO_STRING(THIS^.eActiveCommand);	
END_IF
END_METHOD

{attribute 'monitoring':='call'}
PROPERTY Feedback : I_XP_Feedback
GET
Feedback := THIS^.fbFeedback;
END_GET
END_PROPERTY

(* Calculates which gap the mover should have on a position
	The gap results from the last station crossed.
	If several stations are possible ( switch), the largest gap is displayed here *)
METHOD GapAtPosition : LREAL
VAR_INPUT
	fPosOnTrack : LREAL;//[mm]	
END_VAR
VAR
	ipThisTrack : I_XP_Track := (THIS^);
	bStartAndEndIsOnThisTrack : BOOL;
	ipEachPathOnTrack : I_XP_Path;
END_VAR


THIS^.fbListPathsOnThisTrack.ResetIterator();
WHILE THIS^.fbListPathsOnThisTrack.HasNextObject() DO
	IF __QUERYINTERFACE(THIS^.fbListPathsOnThisTrack.GetNextObject(), ipEachPathOnTrack) THEN
		
		IF ipEachPathOnTrack.Length > ipEachPathOnTrack.DistanceToDestiantion(fPosOnTrack := fPosOnTrack, ipTrack := ipThisTrack) THEN
			GapAtPosition := MAX(GapAtPosition, ipEachPathOnTrack.StationStart.MoverGapAtExit);
		END_IF
			
		//bStartAndEndIsOnThisTrack := ipEachPathOnTrack.StationStart.AccocietedTrack = ipThisTrack AND ipEachPathOnTrack.StationDestination.AccocietedTrack = ipThisTrack; 
		//	
		////Check if start of route is maybe on this track
		//IF (ipEachPathOnTrack.StationStart.AccocietedTrack = ipThisTrack) AND (ipEachPathOnTrack.StationStart.PositionOnTrack > fPosOnTrack) AND NOT bStartAndEndIsOnThisTrack THEN
		//	//start is after the searched position
		//	CONTINUE;
        //
		////Check if end of route is maybe on this track
		//ELSIF (ipEachPathOnTrack.StationDestination.AccocietedTrack = ipThisTrack) AND (ipEachPathOnTrack.StationDestination.PositionOnTrack <= fPosOnTrack) AND NOT bStartAndEndIsOnThisTrack THEN
		//	//end is befor the searched position
		//	CONTINUE;		
		//	
		////Check if in limit - CLOSED LOOP, SHORT SEGMENT Start > End
		//ELSIF F_InLimitTest(fMinimum := ipEachPathOnTrack.StationStart.PositionOnTrack, fInput:= fPosOnTrack, fMaximum := ipEachPathOnTrack.StationDestination.PositionOnTrack) AND bStartAndEndIsOnThisTrack THEN
		//	//track is outside the searched position
		//	CONTINUE;		
        //
		//	
		//ELSE
		//	//The gap is valide, use the largest one
		//	GapAtPosition := MAX(GapAtPosition, ipEachPathOnTrack.StationStart.MoverGapAtExit);
        //
		//END_IF
		
	END_IF
END_WHILE
THIS^.fbListPathsOnThisTrack.RestoreIterator();
END_METHOD

//Each track has an auxiliary station at the end of itself. This is used automatically or not, depending on whether the track also contains stations created by the user.
//These are used by the movers as auxiliary links to navigate through a complex network.
{attribute 'monitoring':='call'}
PROPERTY HelperStationAtEndOfTrack : I_XP_Station
GET
HelperStationAtEndOfTrack :=  THIS^.fbHelpferStationOnEndOfThisTrack;
END_GET
END_PROPERTY

METHOD Initialize : HRESULT
VAR
	hr : HRESULT;
	ipStation : I_XP_Station;
	stVarInfo : __SYSTEM.VAR_INFO;
	sName : STRING;
	ipTcIoXpu : I_TcIoXPlanarProcessingUnit;		
	nIdxXpu : UDINT;
	nIdxTrack : UDINT;
	ipTcIoMover: INT;
END_VAR

VAR_INST
	//This error cannot be reset. Requires a reset cold
	{attribute 'hide'}	
	fbInitError : FB_TcAlarm;
END_VAR
// Check if link to track is mapped
IF NOT THIS^.Mapped THEN
	IF NOT fbInitError.bRaised THEN 
		//This error cannot be reset. Requires a reset cold
		fbInitError.CreateEx(stEventEntry:=TC_EVENTS.CHALET_Base_Events.VariableLinkMissing, ipSourceInfo := THIS^.fbSourceInfo, bWithConfirmation := FALSE);
		stVarInfo := __VARINFO(fbTrack.MCTOPLC_STD);
		fbInitError.ipArguments.AddString(stVarInfo.Symbol);
		fbInitError.Raise(0);
	END_IF
	Initialize := E_FAIL;
	RETURN;
END_IF


IF NOT bInitDone THEN
	//Busy
	Initialize := S_PENDING;
	FW_ObjMgr_GetObjectInstance(oid:= THIS^.fbTrack.MCTOPLC_STD.TrackOID, iid:= TC_GLOBAL_IID_LIST.IID_ITComObject, pipUnk:= ADR(THIS^.ipComObject));	
	
	//TRUE = Use inside PLC the track name from the TcCom Track Object. 
	//FALSE = overwride TcCom Track object with instance name
	IF XPlanarParameterlist.B_TRACK_NAME_TACKOVER_FROM_TRACK_OBJECT THEN
		IF THIS^.ipComObject <> 0 THEN
			THIS^.ipComObject.TcGetObjectName(objName:= ADR(sName), nameLen := SIZEOF(sName));	
			THIS^.fbSourceInfo.sName := sName;
		END_IF
	ELSE
		IF THIS^.ipComObject <> 0 THEN
			sName := THIS^.LUID;
			THIS^.ipComObject.TcSetObjectName(ADR(sName));	
		END_IF
	END_IF
	
	
	//Search interface for this OID
	IF ipXpSystem.Enviroment.UtilityEnvirement <> 0 THEN
		//Get TcIo-Mover interface to utiliy lib
		FOR nIdxTrack := 1 TO Param_TcIoXPlanarEnvironment.MaxXPlanarMoversPerXpu DO
			IF ipXpSystem.Enviroment.UtilityEnvirement.P_TrackOids[nIdxTrack] = THIS^.fbTrack.MCTOPLC_STD.TrackOID THEN
				THIS^.ipUtilityTrack := ipXpSystem.Enviroment.UtilityEnvirement.McTrack(nIdxTrack);
				EXIT;
			END_IF
		END_FOR
	END_IF


	
	//Done as sone list is initilized
	bInitDone := TRUE;
	
ELSE	
	//Done
	Initialize := S_OK;	
END_IF



THIS^.eActiveCommand 				:= CHALET_NC.E_NcAxisCommands.Initialize;
THIS^.fbFeedback.ActiveCommand 		:= TO_STRING(THIS^.eActiveCommand);	
THIS^.fbFeedback.LastCommandAccepted:= TRUE;	
//Set done or keep in busy state	
THIS^.fbFeedback.HR := Initialize;
END_METHOD

{attribute 'monitoring':='call'}
//[mm]
PROPERTY Length : LREAL
GET
Length := THIS^.fbTrack.GetLength();
END_GET
END_PROPERTY

{attribute 'monitoring':='call'}
PROPERTY Mapped : BOOL //Project is mapped to MC (McToPlc and PlcToMc)
GET
VAR
	bMcToPlcNotMapped 	: BOOL;
END_VAR
bMcToPlcNotMapped := F_GetMappingStatus(ADR(THIS^.fbTrack.MCTOPLC_STD), SIZEOF(THIS^.fbTrack.MCTOPLC_STD)) <> EPlcMappingStatus.MS_Mapped;

Mapped := NOT bMcToPlcNotMapped;
END_GET
END_PROPERTY

{attribute 'monitoring':='call'}
//List of interfaces to movers on this track
PROPERTY MoversOnTrack : I_CH_LIST
GET
THIS^.Prepare();//Prepare a list movers on this track


MoversOnTrack := THIS^.fbListOfMoversOnTrack;
END_GET
END_PROPERTY

{attribute 'monitoring':='call'}
// Number of elements describing the geometric curve of the track.
PROPERTY NbOfGeometricElements : UINT
GET
VAR
	nParameterSize : UDINT;
	hr : HRESULT;
	pParaData : PVOID;
	nFoundParameterSize : UDINT;
	nIdx : UDINT;
END_VAR
IF THIS^.ipComObject = 0 THEN
	//Error invalide inteerface
	RETURN;
END_IF

//Read Parameter with an unknown size, repeat until size matches
pParaData := ADR(aRawGeometricElements);
FOR nParameterSize := 0 TO SIZEOF(aRawGeometricElements) BY SIZEOF(aRawGeometricElements[0])  DO 
	
	hr := THIS^.ipComObject.TcGetObjPara(pid:= N_IDX_GEOMETRIC_INFO , nData:= nParameterSize, pData:= pParaData, pgp:=0 );
	
	//Exit if matching size is found
	IF hr = S_OK THEN
		nFoundParameterSize := nParameterSize;
		EXIT;
	END_IF
END_FOR

IF hr <> S_OK THEN
	//Todo Error, list is not matching
	RETURN;
END_IF

//Empty list
IF nFoundParameterSize <= SIZEOF(GUID) THEN
	NbOfGeometricElements := 0;
	RETURN;
END_IF

//Count Nb of GUIDs in raw data
FOR nIdx := 0 TO (nFoundParameterSize-SIZEOF(GUID)) DO
	//Check if at the position x is a GUID of type GUID_MC_POINT_XYC
	IF (Tc2_System.MEMCMP(pBuf1:= ADR(GUID_MC_POINT_XYC), pBuf2:= ADR(aRawGeometricElements[nIdx]), n:= SIZEOF(GUID)) = 0) THEN
		NbOfGeometricElements := NbOfGeometricElements +1;
		nIdx := nIdx + 20; //Skip size of element
	ELSIF (Tc2_System.MEMCMP(pBuf1:= ADR(GUID_MC_LINE_XYC), pBuf2:= ADR(aRawGeometricElements[nIdx]), n:= SIZEOF(GUID)) = 0) THEN
		NbOfGeometricElements := NbOfGeometricElements +1;	
		nIdx := nIdx + 40; //Skip size of element	
	ELSIF (Tc2_System.MEMCMP(pBuf1:= ADR(GUID_MC_CIRCLE_XYC_START_CENTER_END), pBuf2:= ADR(aRawGeometricElements[nIdx]), n:= SIZEOF(GUID)) = 0) THEN
		NbOfGeometricElements := NbOfGeometricElements +1;		
		nIdx := nIdx + 70; //Skip size of element
	END_IF
END_FOR
END_GET
END_PROPERTY

{attribute 'monitoring':='call'}
//Unique object ID
PROPERTY OID : OTCID
GET
OID := THIS^.fbTrack.MCTOPLC_STD.TrackOID;
END_GET
END_PROPERTY

{attribute 'monitoring':='call'}
//List of interfaces to paths on this track
PROPERTY PathsOnTrack : I_CH_List
GET
THIS^.Prepare();//Prepare a list stations on this track

PathsOnTrack := THIS^.fbListPathsOnThisTrack;
END_GET
END_PROPERTY

{attribute 'monitoring':='call'}
PROPERTY PlanarTrack : REFERENCE TO MC_PlanarTrack
GET
PlanarTrack ref= THIS^.fbTrack;
END_GET
END_PROPERTY

(* Time-critical information is processed here, which can then be polled via the property every cycle. 
The update method is usually at the end of the program and then it is already 'outdated'. *)
METHOD PRIVATE Prepare : HRESULT
VAR
	ipThisTrack : I_XP_Track := THIS^;
	ipStation : I_XP_Station;
	ipMover : I_XP_Mover;
	ipPath : I_XP_Path;
END_VAR

VAR_INST
	{attribute 'hide'}
	nLastUpdatedCycleCount : UDINT;
END_VAR
//Check if this Cycle the dates are allready prepared
IF nLastUpdatedCycleCount <> TwinCAT_SystemInfoVarList._TaskInfo[THIS^.nTaskIndex].CycleCount THEN
	nLastUpdatedCycleCount := TwinCAT_SystemInfoVarList._TaskInfo[THIS^.nTaskIndex].CycleCount;

	//Creat a list of all Stations on this Track
	THIS^.fbListOfStationsOnTrack.Clear();
	THIS^.ipXpSystem.StationsUsed.ResetIterator();
	WHILE THIS^.ipXpSystem.StationsUsed.HasNextObject() DO
		IF ToXpStation(THIS^.ipXpSystem.StationsUsed.GetNextObject(), ipStation) AND_THEN ipStation.AccocietedTrack <> 0 AND_THEN ipStation.AccocietedTrack = ipThisTrack THEN
			THIS^.fbListOfStationsOnTrack.AddObject(ipStation);
		END_IF
	END_WHILE
	THIS^.ipXpSystem.StationsUsed.RestoreIterator();
	
	
	
	//Creat a list of all Movers on this Track
	THIS^.fbListOfMoversOnTrack.Clear();
	THIS^.ipXpSystem.MoversPresent.ResetIterator();
	WHILE THIS^.ipXpSystem.MoversPresent.HasNextObject() DO
		IF ToXpMover(THIS^.ipXpSystem.MoversPresent.GetNextObject(), ipMover) AND_THEN ipMover.CurrentTrack <> 0 AND_THEN ipMover.CurrentTrack = ipThisTrack THEN
			THIS^.fbListOfMoversOnTrack.AddObject(ipStation);
		END_IF
	END_WHILE
	THIS^.ipXpSystem.MoversPresent.RestoreIterator();	
	
	
		
	//Creat a list of all Paths on this Track
	THIS^.fbListPathsOnThisTrack.Clear();
	THIS^.ipXpSystem.Paths.ResetIterator();
	WHILE THIS^.ipXpSystem.Paths.HasNextObject() DO
		IF __QUERYINTERFACE(THIS^.ipXpSystem.Paths.GetNextObject(), ipPath)AND_THEN __ISVALIDREF(ipPath.TracksUsed) AND_THEN ipPath.TracksUsed.ObjectInList(ipThisTrack) THEN
			THIS^.fbListPathsOnThisTrack.AddObject(ipPath);
		END_IF
	END_WHILE
	THIS^.ipXpSystem.Paths.RestoreIterator();	
	
END_IF
END_METHOD

METHOD RemoveFromGroup : HRESULT
IF NOT THIS^.fbFeedback.Busy THEN
	THIS^.eActiveCommand 				:= CHALET_NC.E_NcAxisCommands.RemoveFromGroupe;
	THIS^.fbFeedback.ActiveCommand 		:= TO_STRING(THIS^.eActiveCommand);	
	THIS^.fbFeedback.LastCommandAccepted:= TRUE;		
	THIS^.fbFeedback.Busy 				:= TRUE;
	
	THIS^.fbTrack.RemoveFromGroup(THIS^.fbFeedbackRmvFromGrp);
	
	RemoveFromGroup := S_OK;
ELSE
	RemoveFromGroup := S_FALSE;
	THIS^.fbFeedback.LastCommandAccepted:= FALSE;	
END_IF
END_METHOD

//The geometric points of a track are copied. Including the position and type. This only works if the system is disabled.
METHOD ReplicateGeometricElements : HRESULT
VAR_INPUT
	ipTrackCopyFrom : I_XP_Track;
END_VAR
VAR
	ipComObjectExternalTrack  : ITComObject;
	nParameterSize : UDINT;
	hr : HRESULT;
	pParaData : PVOID;
END_VAR
IF THIS^.ipComObject = 0 OR ipTrackCopyFrom = 0 THEN
	//Error invalide interface
	ReplicateGeometricElements := E_HRESULTAdsErr.INVALIDINTERFACE;
	RETURN;
END_IF

pParaData := ADR(aRawGeometricElements);
nParameterSize := SIZEOF(aRawGeometricElements);

//Get interface to external track
hr := FW_ObjMgr_GetObjectInstance(oid:= ipTrackCopyFrom.OID, iid:= TC_GLOBAL_IID_LIST.IID_ITComObject, pipUnk:= ADR(ipComObjectExternalTrack));	

//Read Parameter from external track
IF ipComObjectExternalTrack <> 0 THEN
	hr := ipComObjectExternalTrack.TcGetObjPara(pid:= N_IDX_GEOMETRIC_INFO , nData:= nParameterSize, pData:= pParaData, pgp:=0 );
	
	//Set Parameter in this local track
	IF (hr=S_OK) THEN
		ReplicateGeometricElements := THIS^.ipComObject.TcSetObjPara(pid:= N_IDX_GEOMETRIC_INFO , nData:= nParameterSize, pData:= pParaData, pgp:=0 );
	END_IF
END_IF
END_METHOD

METHOD Reset : HRESULT
VAR_INPUT
END_VAR
THIS^.eActiveCommand 				:= CHALET_NC.E_NcAxisCommands.Reset;
THIS^.fbFeedback.ActiveCommand 		:= TO_STRING(THIS^.eActiveCommand);	
THIS^.fbFeedback.LastCommandAccepted:= TRUE;		
THIS^.fbFeedback.Busy 				:= TRUE;

THIS^.fbTrack.Reset(THIS^.fbFeedbackReset);
Reset := S_OK;
END_METHOD

//move all points of the track geometry. Only works if the system is disabled.
METHOD ShiftTrack : HRESULT
VAR_INPUT
	xOffset, yOffset : LREAL;
END_VAR
VAR
	nParameterSize : UDINT;
	hr : HRESULT;
	pParaData : PVOID;
	nFoundParameterSize : UDINT;
	nIdx : UDINT;
	nTempIndex : UDINT;
END_VAR
IF THIS^.ipComObject = 0 THEN
	//Error invalide interface
	ShiftTrack := E_HRESULTAdsErr.INVALIDINTERFACE;
	RETURN;
END_IF

//Read Parameter with an unknown size, repeat until size matches
pParaData := ADR(aRawGeometricElements);
FOR nParameterSize := 0 TO SIZEOF(aRawGeometricElements) BY SIZEOF(aRawGeometricElements[0])  DO 
	
	hr := THIS^.ipComObject.TcGetObjPara(pid:= N_IDX_GEOMETRIC_INFO , nData:= nParameterSize, pData:= pParaData, pgp:=0 );
	
	//Exit if matching size is found
	IF hr = S_OK THEN
		nFoundParameterSize := nParameterSize;
		EXIT;
	END_IF
END_FOR


//List is not matching
IF hr <> S_OK THEN
	ShiftTrack := Tc2_System.E_HRESULTAdsErr.INVALIDSIZE;
	RETURN;
END_IF

//Empty list
IF nFoundParameterSize <= SIZEOF(GUID) THEN
	ShiftTrack := S_FALSE;
	RETURN;
END_IF

//Count Nb of GUIDs in raw data
FOR nIdx := 0 TO (nFoundParameterSize-SIZEOF(GUID)) DO
	//Check if at the position x is a GUID of type GUID_MC_POINT_XYC
	IF (Tc2_System.MEMCMP(pBuf1:= ADR(GUID_MC_POINT_XYC), pBuf2:= ADR(aRawGeometricElements[nIdx]), n:= SIZEOF(GUID)) = 0) THEN
		//Modify x
		nTempIndex := nIdx+ 2(*GUID*) + 0*1(*LREAL*);
		aRawGeometricElements[nTempIndex] := aRawGeometricElements[nTempIndex] + xOffset;
		//Modify y
		nTempIndex := nIdx+ 2(*GUID*) + 1*1(*LREAL*);
		aRawGeometricElements[nTempIndex] := aRawGeometricElements[nTempIndex] + yOffset;
		nIdx := nIdx + 3 -1; //Skip size of element
	ELSIF (Tc2_System.MEMCMP(pBuf1:= ADR(GUID_MC_LINE_XYC), pBuf2:= ADR(aRawGeometricElements[nIdx]), n:= SIZEOF(GUID)) = 0) THEN
		//Modify start x
		nTempIndex := nIdx+ 2(*GUID*) + 0*1(*LREAL*);
		aRawGeometricElements[nTempIndex] := aRawGeometricElements[nTempIndex] + xOffset;
		//Modify start y
		nTempIndex := nIdx+ 2(*GUID*) + 1*1(*LREAL*);
		aRawGeometricElements[nTempIndex] := aRawGeometricElements[nTempIndex] + yOffset;
		//Modify end x
		nTempIndex := nIdx+ 2(*GUID*) + 3*1(*LREAL*);
		aRawGeometricElements[nTempIndex] := aRawGeometricElements[nTempIndex] + xOffset;
		//Modify end y
		nTempIndex := nIdx+ 2(*GUID*) + 4*1(*LREAL*);
		aRawGeometricElements[nTempIndex] := aRawGeometricElements[nTempIndex] + yOffset;
		nIdx := nIdx + 6 -1; //Skip size of element	
	ELSIF (Tc2_System.MEMCMP(pBuf1:= ADR(GUID_MC_CIRCLE_XYC_START_CENTER_END), pBuf2:= ADR(aRawGeometricElements[nIdx]), n:= SIZEOF(GUID)) = 0) THEN
		//Modify start x
		nTempIndex := nIdx+ 2(*GUID*) + 0*1(*LREAL*);
		aRawGeometricElements[nTempIndex] := aRawGeometricElements[nTempIndex] + xOffset;
		//Modify start y
		nTempIndex := nIdx+ 2(*GUID*) + 1*1(*LREAL*);
		aRawGeometricElements[nTempIndex] := aRawGeometricElements[nTempIndex] + yOffset;
		//Modify end x
		nTempIndex := nIdx+ 2(*GUID*) + 3*1(*LREAL*);
		aRawGeometricElements[nTempIndex] := aRawGeometricElements[nTempIndex] + xOffset;
		//Modify end y
		nTempIndex := nIdx+ 2(*GUID*) + 4*1(*LREAL*);
		aRawGeometricElements[nTempIndex] := aRawGeometricElements[nTempIndex] + yOffset;
		//Modify center x
		nTempIndex := nIdx+ 2(*GUID*) + 6*1(*LREAL*);
		aRawGeometricElements[nTempIndex] := aRawGeometricElements[nTempIndex] + xOffset;
		//Modify center y
		nTempIndex := nIdx+ 2(*GUID*) + 7*1(*LREAL*);
		aRawGeometricElements[nTempIndex] := aRawGeometricElements[nTempIndex] + yOffset;
		nIdx := nIdx + 9 -1; //Skip size of element
	END_IF
END_FOR


//Write new raw parameter to tccom track
pParaData := ADR(aRawGeometricElements);
ShiftTrack := THIS^.ipComObject.TcSetObjPara(pid:= N_IDX_GEOMETRIC_INFO , nData:= nFoundParameterSize, pData:= pParaData, pgp:=0 );
END_METHOD

{attribute 'monitoring':='call'}
//Position of the start point of this tracks
PROPERTY StartPosition : REFERENCE TO MoverVector
GET
VAR_INST
	stStartPositionXY : MoverVector;
END_VAR
VAR
	fbPositionXYC : PositionXYC;
END_VAR
THIS^.fbTrack.GetPositionAt(0,position := fbPositionXYC);


stStartPositionXY.x := fbPositionXYC.x;
stStartPositionXY.y := fbPositionXYC.y;
stStartPositionXY.z := 0;
stStartPositionXY.a := 0;
stStartPositionXY.b := 0;
stStartPositionXY.c := fbPositionXYC.c;



StartPosition REF= stStartPositionXY;
END_GET
END_PROPERTY

(* Returns the first station on current track who has exact thsi position or is ahead
	If no station on this track, result is maybe on another track*)
METHOD StationAhedPosition : I_XP_Station
VAR_INPUT
	fPosOnTrack : LREAL;//[mm]	
END_VAR
VAR
	fDistToTempBestStaton : LREAL := CHALET_BaseComponents.GVL_Datatypes.cMaxLreal;;
	ipTempBestStation : I_XP_Station;
	fDist :LREAL;
	bStartAndEndIsOnThisTrack : BOOL;
	ipThisTrack : I_XP_Track := (THIS^);
	ipEachPathOnTrack : I_XP_Path;
END_VAR
THIS^.fbListPathsOnThisTrack.ResetIterator();
WHILE THIS^.fbListPathsOnThisTrack.HasNextObject() DO
	IF __QUERYINTERFACE(THIS^.fbListPathsOnThisTrack.GetNextObject(), ipEachPathOnTrack) THEN
		
		bStartAndEndIsOnThisTrack := ipEachPathOnTrack.StationStart.AccocietedTrack = ipThisTrack AND ipEachPathOnTrack.StationDestination.AccocietedTrack = ipThisTrack; 
		
		//Check if end of route is not before this station
		IF (ipEachPathOnTrack.StationDestination.AccocietedTrack = ipThisTrack) AND (ipEachPathOnTrack.StationDestination.PositionOnTrack < fPosOnTrack) AND NOT bStartAndEndIsOnThisTrack THEN
			//end is before the searched position - not a valide target
			CONTINUE;		
		END_IF
		
		//Check if end of route is before this station - CLOSED LOOP, SHORT SEGMENT
		IF NOT F_InLimitTest(fMinimum := ipEachPathOnTrack.StationStart.PositionOnTrack, fInput:= fPosOnTrack, fMaximum := ipEachPathOnTrack.StationDestination.PositionOnTrack) AND bStartAndEndIsOnThisTrack THEN
			//end is before the searched position - not a valide target
			CONTINUE;		
		END_IF
	
			
		fDist := ipEachPathOnTrack.DistanceToDestiantion(	ipTrack := ipThisTrack, 
															fPosOnTrack := 	fPosOnTrack);
															
		//Get shortest distance													
		IF 	fDist <= fDistToTempBestStaton	THEN
			fDistToTempBestStaton := fDist;
			ipTempBestStation := ipEachPathOnTrack.StationDestination;
		END_IF
		
	END_IF
END_WHILE
THIS^.fbListPathsOnThisTrack.RestoreIterator();

StationAhedPosition := ipTempBestStation;
END_METHOD

(* Returns the first station on current track who has exact thsi position or is behind
	If no station on this track, result is maybe on another track*)
METHOD StationBehindPosition : I_XP_Station
VAR_INPUT
	fPosOnTrack : LREAL;//[mm]	
END_VAR
VAR
	fDistToTempBestStaton : LREAL := CHALET_BaseComponents.GVL_Datatypes.cMaxLreal;;
	ipTempBestStation : I_XP_Station;
	fDist :LREAL;
	bStartAndEndIsOnThisTrack : BOOL;
	ipThisTrack : I_XP_Track := (THIS^);
	ipEachPathOnTrack : I_XP_Path;
END_VAR
THIS^.fbListPathsOnThisTrack.ResetIterator();
WHILE THIS^.fbListPathsOnThisTrack.HasNextObject() DO
	IF __QUERYINTERFACE(THIS^.fbListPathsOnThisTrack.GetNextObject(), ipEachPathOnTrack) THEN
		
		bStartAndEndIsOnThisTrack := ipEachPathOnTrack.StationStart.AccocietedTrack = ipThisTrack AND ipEachPathOnTrack.StationDestination.AccocietedTrack = ipThisTrack; 
		
		//Check if end of route is not before this station
		IF (ipEachPathOnTrack.StationDestination.AccocietedTrack = ipThisTrack) AND (ipEachPathOnTrack.StationDestination.PositionOnTrack < fPosOnTrack) AND NOT bStartAndEndIsOnThisTrack THEN
			//end is before the searched position - not a valide target
			CONTINUE;		
		END_IF
		
		//Check if end of route is before this station - CLOSED LOOP, SHORT SEGMENT
		IF NOT F_InLimitTest(fMinimum := ipEachPathOnTrack.StationStart.PositionOnTrack, fInput:= fPosOnTrack, fMaximum := ipEachPathOnTrack.StationDestination.PositionOnTrack) AND bStartAndEndIsOnThisTrack THEN
			//end is before the searched position - not a valide target
			CONTINUE;		
		END_IF
	
		//Dist to Start	
		fDist := ipEachPathOnTrack.Length - ipEachPathOnTrack.DistanceToDestiantion(	ipTrack := ipThisTrack, 
																						fPosOnTrack := 	fPosOnTrack);
															
		//Get shortest distance													
		IF 	fDist <= fDistToTempBestStaton	THEN
			fDistToTempBestStaton := fDist;
			ipTempBestStation := ipEachPathOnTrack.StationDestination;
		END_IF
		
	END_IF
END_WHILE
THIS^.fbListPathsOnThisTrack.RestoreIterator();

StationBehindPosition := ipTempBestStation;
END_METHOD

(* Returns the closest station on current, ahead or behind track*)
METHOD StationClosestTo : I_XP_Station
VAR_INPUT
	fPosOnTrack : LREAL;//[mm]	
END_VAR
VAR
	fDistToTempBestStaton : LREAL := CHALET_BaseComponents.GVL_Datatypes.cMaxLreal;;
	ipTempBestStation : I_XP_Station;
	fDist :LREAL;
	bStartAndEndIsOnThisTrack : BOOL;
	ipThisTrack : I_XP_Track := (THIS^);
	ipEachPathOnTrack : I_XP_Path;
END_VAR
THIS^.fbListPathsOnThisTrack.ResetIterator();
WHILE THIS^.fbListPathsOnThisTrack.HasNextObject() DO
	IF __QUERYINTERFACE(THIS^.fbListPathsOnThisTrack.GetNextObject(), ipEachPathOnTrack) THEN
		
		bStartAndEndIsOnThisTrack := ipEachPathOnTrack.StationStart.AccocietedTrack = ipThisTrack AND ipEachPathOnTrack.StationDestination.AccocietedTrack = ipThisTrack; 
		
		//Check if end of route is not before this station
		IF (ipEachPathOnTrack.StationDestination.AccocietedTrack = ipThisTrack) AND (ipEachPathOnTrack.StationDestination.PositionOnTrack < fPosOnTrack) AND NOT bStartAndEndIsOnThisTrack THEN
			//end is before the searched position - not a valide target
			CONTINUE;		
		END_IF
		
		//Check if end of route is before this station - CLOSED LOOP, SHORT SEGMENT
		IF NOT F_InLimitTest(fMinimum := ipEachPathOnTrack.StationStart.PositionOnTrack, fInput:= fPosOnTrack, fMaximum := ipEachPathOnTrack.StationDestination.PositionOnTrack) AND bStartAndEndIsOnThisTrack THEN
			//end is before the searched position - not a valide target
			CONTINUE;		
		END_IF
	
		//Dist to End				
		fDist := ipEachPathOnTrack.DistanceToDestiantion(	ipTrack := ipThisTrack, 
															fPosOnTrack := 	fPosOnTrack);
		//Dist to Start	
		fDist := MIN(fDist, ipEachPathOnTrack.Length - ipEachPathOnTrack.DistanceToDestiantion(	ipTrack := ipThisTrack, 
																						fPosOnTrack := 	fPosOnTrack));


															
		//Get shortest distance													
		IF 	fDist <= fDistToTempBestStaton	THEN
			fDistToTempBestStaton := fDist;
			ipTempBestStation := ipEachPathOnTrack.StationDestination;
		END_IF
		
	END_IF
END_WHILE
THIS^.fbListPathsOnThisTrack.RestoreIterator();

StationClosestTo := ipTempBestStation;
END_METHOD

{attribute 'monitoring':='call'}
//List of interfaces to stations on this track
PROPERTY StationsOnTrack : I_CH_List
GET
THIS^.Prepare();//Prepare a list stations on this track

StationsOnTrack := THIS^.fbListOfStationsOnTrack;
END_GET
END_PROPERTY

{attribute 'monitoring':='call'}
//Interface to CHALET system to which this object belongs
PROPERTY System : I_XP_System_PLC
GET
//get I_x_System_PLC interface from I_x_System_Registration
__QUERYINTERFACE(THIS^.ipXpSystem, System);
END_GET
END_PROPERTY

{attribute 'monitoring':='call'}
//List of interfaces from other tracks
PROPERTY TracksAhead : I_CH_List
GET
TracksAhead := fbTracksAhead;
END_GET
END_PROPERTY

{attribute 'monitoring':='call'}
//List of interfaces from other tracks
PROPERTY TracksBehinde : I_CH_List
GET
TracksBehinde:= fbTracksBehinde;
END_GET
END_PROPERTY

{attribute 'monitoring':='call'}
//zzz Todo Delet me
PROPERTY TracksEndAtThis : REFERENCE TO  ARRAY[0..(XPlanarParameterlist.N_MAX_STATIONS_AHEAD_OR_BEHIND-1)] OF I_XP_Track
GET
TracksEndAtThis REF= ipTracksEndAtThis;
END_GET
END_PROPERTY

{attribute 'monitoring':='call'}
PROPERTY TracksStartFromThis : REFERENCE TO ARRAY[0..(XPlanarParameterlist.N_MAX_STATIONS_AHEAD_OR_BEHIND-1)] OF I_XP_Track
GET
TracksStartFromThis REF= ipTracksStartFromThis;
END_GET
END_PROPERTY

METHOD PUBLIC Update : HRESULT
VAR_INPUT
END_VAR

THIS^.Prepare();//Prepare time-critical information, if not already done



// ********************** Set feedback depending on active command *******************************
CASE THIS^.eActiveCommand OF
	E_NcAxisCommands.None: 
		//Display if a Mover Error is active during no command is active
		IF THIS^.fbTrack.Error AND NOT fbFeedback.Error THEN 
			fbFeedback.ErrorId 			:= THIS^.fbTrack.ErrorID;
			fbFeedback.ActiveCommand 	:= TO_STRING(E_NcAxisCommands.None);	
			fbFeedback.ClearObjectInfo();
		END_IF

	E_NcAxisCommands.Initialize:
		fbFeedback.Busy 			:= NOT THIS^.bInitDone;
		fbFeedback.Done 			:= THIS^.bInitDone;
		fbFeedback.ErrorId 			:= 0;
		fbFeedback.ClearObjectInfo();
		                        	
	E_NcAxisCommands.Enable:     	
		fbFeedback.Busy 			:= fbFeedbackEnable.Busy;
		fbFeedback.Done 			:= fbFeedbackEnable.Done;
		fbFeedback.ErrorId 			:= fbFeedbackEnable.ErrorID;
        fbFeedback.ObjectInfo		:= fbFeedbackEnable.objectInfo;
                                			                        	
	E_NcAxisCommands.Disable:     	
		fbFeedback.Busy 			:= fbFeedbackDisable.Busy;
		fbFeedback.Done 			:= fbFeedbackDisable.Done;
		fbFeedback.ErrorId 			:= fbFeedbackDisable.ErrorID;
        fbFeedback.ObjectInfo		:= fbFeedbackDisable.objectInfo;
		
	E_NcAxisCommands.Configure:
		fbFeedback.Busy 		:= nSeqConfiguring > 0;
		fbFeedback.Done 		:= nSeqConfiguring = 999;
		IF nSeqConfiguring > 1000 THEN
			fbFeedback.ErrorId 		:= nSeqConfiguring;
		END_IF
                                			                        	
	E_NcAxisCommands.Reset:     	
		fbFeedback.Busy 			:= fbFeedbackReset.Busy;
		fbFeedback.Done 			:= fbFeedbackReset.Done;
		fbFeedback.ErrorId 			:= fbFeedbackReset.ErrorID;
        fbFeedback.ObjectInfo		:= fbFeedbackReset.objectInfo;
                                      			                        	
	E_NcAxisCommands.AddToGroupe:     	
		fbFeedback.Busy 			:= fbFeedbackAddToGrp.Busy;
		fbFeedback.Done 			:= fbFeedbackAddToGrp.Done;
		fbFeedback.ErrorId 			:= fbFeedbackAddToGrp.ErrorID;
        fbFeedback.ObjectInfo		:= fbFeedbackAddToGrp.objectInfo;
                                      			                        	
	E_NcAxisCommands.RemoveFromGroupe:     	
		fbFeedback.Busy 			:= fbFeedbackRmvFromGrp.Busy;
		fbFeedback.Done 			:= fbFeedbackRmvFromGrp.Done;
		fbFeedback.ErrorId 			:= fbFeedbackRmvFromGrp.ErrorID;
        fbFeedback.ObjectInfo		:= fbFeedbackRmvFromGrp.objectInfo;
                                		
	ELSE//External command in subclass
		;
END_CASE


// **********************  Stop to execute commands on .done or .error ***************************
IF fbFeedback.Done OR THIS^.fbFeedback.Error THEN
	eActiveCommand 				:= E_NcAxisCommands.None;
END_IF

//Update xplanar object
THIS^.fbTrack.Update();

//Update feedback object
fbFeedbackEnable.Update(); 
fbFeedbackDisable.Update(); 
fbFeedbackReset.Update(); 
fbFeedbackAddToGrp.Update(); 
fbFeedbackRmvFromGrp.Update();
END_METHOD

{attribute 'monitoring':='call'}
//Interface to this track in XPlanar Utility Lib
PROPERTY UtilityTrack : Tc3_XPlanarUtility.I_McPlanarTrack
GET
UtilityTrack :=  THIS^.ipUtilityTrack;
END_GET
END_PROPERTY

END_FUNCTION_BLOCK
